// TIA Portal V18 export
// export: Created 2026-01-09T11:32:03.7635305Z, ExportSetting WithDefaults, DisplayName Totally Integrated Automation Portal, DisplayVersion V18 Update 5, DisplayName TIA Portal Openness, DisplayVersion V18 Update 5, DisplayName TIA Portal Teamcenter Gateway, DisplayVersion V18, DisplayName TIA Portal Version Control Interface, DisplayVersion V18, DisplayName SINAMICS Startdrive Advanced, DisplayVersion V18 SP2 Update 1, DisplayName SINAMICS Startdrive G110M, G120, G120C, G120D, G120P, G115D, DisplayVersion V18 SP2 Update 1, DisplayName SINAMICS Startdrive G130, G150, S120, S150, SINAMICS MV, S210, G220, S200, DisplayVersion V18 SP2 Update 1, DisplayName STEP 7 Professional, DisplayVersion V18 Update 5, DisplayName STEP 7 Safety, DisplayVersion V18, DisplayName WinCC Professional, DisplayVersion V18 Update 5
TagTable "ST_CycleTime"
  ST_MachineCycleTimeNo[0] : Real  (%DB[ST_SysDBNum].DBD600, CPU S71500-2PN_TP700, 1 s)
  ST_MachineCycleTimeNo[01] : Real  (%DB[ST_SysDBNum].DBD604, CPU S71500-2PN_TP700, 1 s)
  ST_MachineCycleTimeNo[02] : Real  (%DB[ST_SysDBNum].DBD608, CPU S71500-2PN_TP700, 1 s)
  ST_MachineCycleTimeNo[03] : Real  (%DB[ST_SysDBNum].DBD612, CPU S71500-2PN_TP700, 1 s)
  ST_MachineCycleTimeNo[04] : Real  (%DB[ST_SysDBNum].DBD616, CPU S71500-2PN_TP700, 1 s)
  ST_MachineCycleTimeNo[05] : Real  (%DB[ST_SysDBNum].DBD620, CPU S71500-2PN_TP700, 1 s)
  ST_MachineCycleTimeNo[06] : Real  (%DB[ST_SysDBNum].DBD624, CPU S71500-2PN_TP700, 1 s)
  ST_MachineCycleTimeNo[07] : Real  (%DB[ST_SysDBNum].DBD628, CPU S71500-2PN_TP700, 1 s)
  ST_MachineCycleTimeNo[08] : Real  (%DB[ST_SysDBNum].DBD632, CPU S71500-2PN_TP700, 1 s)
  ST_MachineCycleTimeNo[09] : Real  (%DB[ST_SysDBNum].DBD636, CPU S71500-2PN_TP700, 1 s)
  ST_MachineCycleTimeNo[10] : Real  (%DB[ST_SysDBNum].DBD640, CPU S71500-2PN_TP700, 1 s)
  ST_MachineCycleTimeNo[11] : Real  (%DB[ST_SysDBNum].DBD644, CPU S71500-2PN_TP700, 1 s)
  ST_MachineCycleTimeNo[12] : Real  (%DB[ST_SysDBNum].DBD648, CPU S71500-2PN_TP700, 1 s)
  ST_MachineCycleTimeNo[13] : Real  (%DB[ST_SysDBNum].DBD652, CPU S71500-2PN_TP700, 1 s)
  ST_MachineCycleTimeNo[14] : Real  (%DB[ST_SysDBNum].DBD656, CPU S71500-2PN_TP700, 1 s)
  ST_MachineCycleTimeNo[15] : Real  (%DB[ST_SysDBNum].DBD660, CPU S71500-2PN_TP700, 1 s)
  ST_MachineCycleTimeNo[16] : Real  (%DB[ST_SysDBNum].DBD664, CPU S71500-2PN_TP700, 1 s)
  ST_MachineCycleTimeNo[17] : Real  (%DB[ST_SysDBNum].DBD668, CPU S71500-2PN_TP700, 1 s)
  ST_MachineCycleTimeNo[18] : Real  (%DB[ST_SysDBNum].DBD672, CPU S71500-2PN_TP700, 1 s)
  ST_MachineCycleTimeNo[19] : Real  (%DB[ST_SysDBNum].DBD676, CPU S71500-2PN_TP700, 1 s)
  ST_MachineCycleTimeNo[20] : Real  (%DB[ST_SysDBNum].DBD680, CPU S71500-2PN_TP700, 1 s)
  ST_MachineCycleTimeNo[21] : Real  (%DB[ST_SysDBNum].DBD684, CPU S71500-2PN_TP700, 1 s)
  ST_TotalCycleTimeNo[0] : Real  (%DB[ST_SysDBNum].DBD500, CPU S71500-2PN_TP700, 1 s)
  ST_TotalCycleTimeNo[01] : Real  (%DB[ST_SysDBNum].DBD504, CPU S71500-2PN_TP700, 1 s)
  ST_TotalCycleTimeNo[02] : Real  (%DB[ST_SysDBNum].DBD508, CPU S71500-2PN_TP700, 1 s)
  ST_TotalCycleTimeNo[03] : Real  (%DB[ST_SysDBNum].DBD512, CPU S71500-2PN_TP700, 1 s)
  ST_TotalCycleTimeNo[04] : Real  (%DB[ST_SysDBNum].DBD516, CPU S71500-2PN_TP700, 1 s)
  ST_TotalCycleTimeNo[05] : Real  (%DB[ST_SysDBNum].DBD520, CPU S71500-2PN_TP700, 1 s)
  ST_TotalCycleTimeNo[06] : Real  (%DB[ST_SysDBNum].DBD524, CPU S71500-2PN_TP700, 1 s)
  ST_TotalCycleTimeNo[07] : Real  (%DB[ST_SysDBNum].DBD528, CPU S71500-2PN_TP700, 1 s)
  ST_TotalCycleTimeNo[08] : Real  (%DB[ST_SysDBNum].DBD532, CPU S71500-2PN_TP700, 1 s)
  ST_TotalCycleTimeNo[09] : Real  (%DB[ST_SysDBNum].DBD536, CPU S71500-2PN_TP700, 1 s)
  ST_TotalCycleTimeNo[10] : Real  (%DB[ST_SysDBNum].DBD540, CPU S71500-2PN_TP700, 1 s)
  ST_TotalCycleTimeNo[11] : Real  (%DB[ST_SysDBNum].DBD544, CPU S71500-2PN_TP700, 1 s)
  ST_TotalCycleTimeNo[12] : Real  (%DB[ST_SysDBNum].DBD548, CPU S71500-2PN_TP700, 1 s)
  ST_TotalCycleTimeNo[13] : Real  (%DB[ST_SysDBNum].DBD552, CPU S71500-2PN_TP700, 1 s)
  ST_TotalCycleTimeNo[14] : Real  (%DB[ST_SysDBNum].DBD556, CPU S71500-2PN_TP700, 1 s)
  ST_TotalCycleTimeNo[15] : Real  (%DB[ST_SysDBNum].DBD560, CPU S71500-2PN_TP700, 1 s)
  ST_TotalCycleTimeNo[16] : Real  (%DB[ST_SysDBNum].DBD564, CPU S71500-2PN_TP700, 1 s)
  ST_TotalCycleTimeNo[17] : Real  (%DB[ST_SysDBNum].DBD568, CPU S71500-2PN_TP700, 1 s)
  ST_TotalCycleTimeNo[18] : Real  (%DB[ST_SysDBNum].DBD572, CPU S71500-2PN_TP700, 1 s)
  ST_TotalCycleTimeNo[19] : Real  (%DB[ST_SysDBNum].DBD576, CPU S71500-2PN_TP700, 1 s)
  ST_TotalCycleTimeNo[20] : Real  (%DB[ST_SysDBNum].DBD580, CPU S71500-2PN_TP700, 1 s)
  ST_TotalCycleTimeNo[21] : Real  (%DB[ST_SysDBNum].DBD584, CPU S71500-2PN_TP700, 1 s)
